// Mitsubishi GX Works2 project: b04   PLC: Q02/Q02H

PROGRAM MAIN
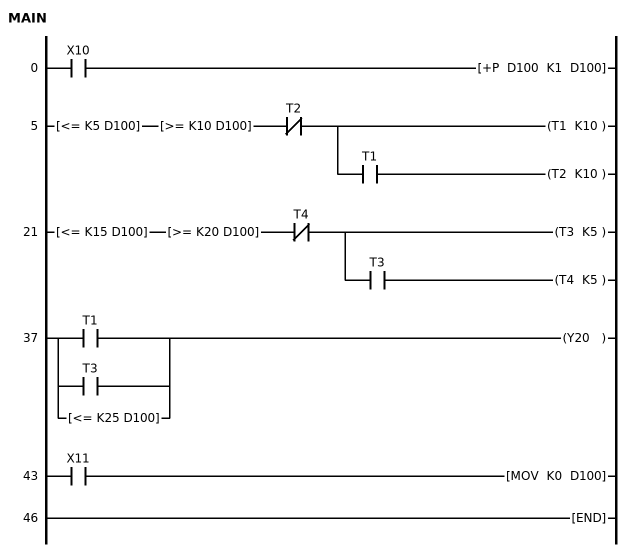
0     LD      X10
      +P      D100 K1 D100
5     LD<=    K5 D100
      AND>=   K10 D100
      ANI     T2
      OUT     T1 K10
      AND     T1
      OUT     T2 K10
21    LD<=    K15 D100
      AND>=   K20 D100
      ANI     T4
      OUT     T3 K5
      AND     T3
      OUT     T4 K5
37    LD      T1
      OR      T3
      OR<=    K25 D100
      OUT     Y20
43    LD      X11
      MOV     K0 D100
46    END
END_PROGRAM
